(* CODESYS project AxisControl.export

Project tree, tasks and I/O mapping:
  AxisControl/
    data type MutiAxisMoveMethod
    function block AuxAxis_PowerOn [ST]
    function block MultiAxisABSMove [ST]
    function block MultiAxisTorqueLimit [ST]
*)

// AxisControl/MutiAxisMoveMethod
TYPE MutiAxisMoveMethod :
(
	None := 0				// all axis move at same vel as given
	, SpeedControl := 10		// all axis arrive destination at same time
);
END_TYPE

// AxisControl/AuxAxis_PowerOn
FUNCTION_BLOCK AuxAxis_PowerOn
VAR_INPUT
	Enable : BOOL;
END_VAR
VAR_OUTPUT
	Done : BOOL;
	Error : BOOL;
	Err_Message : Error_Message;
END_VAR
VAR
	_state : INT := 0;
	_end : BOOL := TRUE;
	_Timer: ton;
	_err_time : TIME := T#5S;
	
	// read cfg message
	ReadCfg : ArcaLibrary.SYS_GetConfigInfo;
	Num_of_Axis:WORD;
	Num_of_Groups:WORD;
	Num_of_Cams:WORD;
	MotionCfgOK: BOOL;
	ECatCfgOk: BOOL;
	VisionCfgOk: BOOL;
	
	// power settings
	PowBlk:ARRAY[1..48] OF ArcaLibrary.MC_Power;
	PowDone, PowErr: ARRAY [1..48] OF BOOL;
	power_On_States : INT := 0;
	All_Power_On_Check_Counter : INT;
	Power_Err_Check_Counter : INT;
	Power_Counter : INT;
	
	//reset blocks
	AxRes:ARRAY[1..48] OF ArcaLibrary.MC_Reset;
	AxResDone, AxResErr: ARRAY [1..48] OF BOOL;
	rest_counter : INT := 0;
	All_reset_On : BOOL;
	All_reset_On_Check_Counter : INT;
	reset_Err_Check_Counter : INT;
	reset_State : INT := 0;
	
	//group management
	GrpEn: ARRAY[1..5] OF ArcaLibrary.MC_GroupEnable;
	GrpDis: ARRAY[1..5] OF ArcaLibrary.MC_GroupDisable;
	GrpErr : ARRAY [1..5] OF BOOL;
	Grp_En_State : INT;
	Grp_counter : INT;
	Grp_En_Check_Counter : INT;
	Grp_Dis_Counter : INT;
	
	//debug
END_VAR

IF enable  THEN
	_end := FALSE;
ELSE
	_state := -10;
END_IF

IF _end = TRUE THEN
	RETURN;
END_IF

_Timer(in:= (power_On_States = 10) OR (reset_State = 10) OR (Grp_En_State = 10), pt:= _err_time);

// read how many axis has been config
ReadCfg(axisnumber => Num_of_axis, groupnumber => Num_of_Groups, cameranumber => Num_of_Cams
	, MotionCfgOk => MotionCfgOK, ecatcfgok => ECatCfgOk, visioncfgok => VisionCfgOk);

// power blocks
CASE (power_On_States) OF
	0:	
		IF (_state>0 AND _state<100) AND ECatCfgOk AND MotionCfgOK THEN
			power_On_States := 10;
		END_IF
	10:
		All_Power_On_Check_Counter := 1;
		FOR Power_Counter:=1 TO WORD_TO_INT(Num_of_axis) DO
			PowBlk[Power_Counter](Axis:=Power_Counter -1, Enable:=TRUE, EnablePositive:=TRUE, EnableNegative:=TRUE, Status=>PowDone[Power_Counter], Error=>PowErr[Power_Counter]);
			IF PowDone[Power_Counter] = TRUE THEN
				All_Power_On_Check_Counter := All_Power_On_Check_Counter + 1;
			END_IF
		END_FOR
		
		IF All_Power_On_Check_Counter >= WORD_TO_INT(Num_of_axis) THEN
			power_On_States := 20;
		ELSIF _Timer.Q THEN
			_state := -21;
		END_IF
		IF (_state<=0 OR _state>=100) THEN
			power_On_States := 30;
		END_IF
	20:
		IF (_state<=0 OR _state>=100) THEN
			power_On_States := 30;
		END_IF
	30:
		FOR Power_Counter:=1 TO WORD_TO_INT(Num_of_axis) DO
			PowBlk[Power_Counter](Axis:=Power_Counter -1, Enable:=FALSE);
		END_FOR
		power_On_States := 0;
END_CASE
// check if power block is err
IF power_On_States > 0 AND power_On_States < 30 THEN
	FOR Power_Err_Check_Counter:=1 TO WORD_TO_INT(Num_of_axis) DO
			IF PowBlk[Power_Err_Check_Counter - 1].Error = TRUE THEN
				//_state := -20;
			END_IF
	END_FOR
END_IF

// reset blocks
CASE (reset_State) OF
	0:
		All_reset_On := FALSE;
		IF _state=2 THEN
			reset_state := 10;
		END_IF
	10:
		All_reset_On_Check_Counter := 0;
		FOR rest_counter:=1 TO WORD_TO_INT(Num_of_axis) DO
			AxRes[rest_counter](Axis:=rest_counter - 1, Execute:=TRUE, Done=>AxResDone[rest_counter], Error=>AxResErr[rest_counter]);
			IF AxRes[rest_counter].Done = TRUE THEN
				All_reset_On_Check_Counter := All_reset_On_Check_Counter +1;
			END_IF
		END_FOR
		IF All_reset_On_Check_Counter = WORD_TO_INT(Num_of_axis) THEN
			All_reset_On := TRUE;
		ELSIF _Timer.Q THEN
			_state := -31;
		END_IF
		IF (_state <> 2) THEN
			reset_State := 0;
		END_IF
END_CASE
// check if reset block is err
IF reset_State <> 0 THEN
	FOR reset_Err_Check_Counter:=1 TO WORD_TO_INT(Num_of_axis) DO
			IF AxRes[reset_Err_Check_Counter - 1].Error = TRUE THEN
				_state := -30;
			END_IF
	END_FOR
END_IF

// group enable/disable
CASE Grp_En_State OF
	0:
		IF _state >= 30 AND _state <=100 THEN
			grp_counter := 1;
			Grp_En_State := 10;
		END_IF
	10:	
		IF grp_counter > WORD_TO_INT(Num_of_Groups) THEN
			Grp_En_State := 20;
		ELSE
			GrpEn[grp_counter](AxesGroup := grp_counter - 1, Execute := TRUE);
			IF GrpEn[grp_counter].Done THEN
				IF grp_counter <= WORD_TO_INT(Num_of_Groups) THEN
					grp_counter := grp_counter +1;
				END_IF
			ELSIF _Timer.Q THEN
				_state := -41;
			END_IF
		END_IF
		
		IF (_state < 30 OR _state > 100) THEN
			Grp_En_State := 30;
		END_IF
	20:
		IF (_state < 30 OR _state > 100) THEN
			Grp_En_State := 30;
		END_IF
	30:
		FOR grp_counter := 1 TO WORD_TO_INT(Num_of_Groups) DO
			GrpEn[grp_counter](AxesGroup := grp_counter - 1, Execute := FALSE);
		END_FOR
		Grp_En_State := 0;
	
END_CASE
// check if enable block is err
IF Grp_En_State = 9990 THEN
	FOR Grp_En_Check_Counter:=1 TO WORD_TO_INT(Num_of_Groups) DO
			IF GrpEn[Grp_En_Check_Counter - 1].Error = TRUE THEN
				_state := -40;
			END_IF
	END_FOR
END_IF

// disable group when all group enable block are off
FOR Grp_Dis_Counter := 1 TO WORD_TO_INT(Num_of_Groups) DO
	GrpDis[Grp_Dis_Counter](AxesGroup:= Grp_Dis_Counter - 1, Execute:= Grp_En_State = 0);
END_FOR

//	manager
CASE _state OF
	-41:
		error := TRUE;
		err_message := Error_Message.Err_Group_Enable_TimeOut;
	-40:
		error := TRUE;
		err_message := Error_Message.Err_Group_Enable_Block_Err;
		
	-31:
		error := TRUE;
		err_message := Error_Message.Err_Power_Reset_TimeOut;
	-30:
		error := TRUE;
		err_message := Error_Message.Err_Power_Reset_Block_Err;
		
	-21:
		error := TRUE;
		err_message := Error_Message.Err_PowerOn_TimeOut;
	-20:
		error := TRUE;
		err_message := Error_Message.Err_PowerOn_Block_Err;
	-10:
		IF power_On_States = 0 AND reset_State = 0 AND Grp_En_State = 0 THEN
			done := error := FALSE;
			err_message := error_message.Err_None;
			_end := TRUE;
			_state := 0;
		END_IF
	0:
		IF enable AND power_On_States = 0 AND reset_State = 0 AND Grp_En_State = 0 THEN
			_state := 10;
		END_IF
	10:
		IF power_On_States = 20 THEN
			_state := 30;
		END_IF
	30:
		IF Grp_En_State = 20 THEN
			_state := 40;
		END_IF
	40:
		done := TRUE;
END_CASE

END_FUNCTION_BLOCK

// AxisControl/MultiAxisABSMove
FUNCTION_BLOCK MultiAxisABSMove
VAR_INPUT
	FirstAuxAxisNum : BYTE;	// for safty reason, this block do not accept different axis after enabled
	LastAuxAxisNum : BYTE;
	Enable : BOOL;
	Axis_Mov_Indicator : ARRAY [0..255] OF BOOL; // tell program which axis to mov whih not mov
	Axis_Mov_Pos : ARRAY [0..255] OF REAL; // tell program which axis to what position
	Execute : BOOL;
	Vel, Acc, Dec, Jerk : REAL;	// not allow 0 or none input
	MoveMethod : MutiAxisMoveMethod;
END_VAR
VAR_OUTPUT
	done : BOOL;
	error : BOOL;
	error_str : STRING;
END_VAR
VAR
	_Faxis, _Laxis : BYTE;	// internal first axis and last axis
	_Indicator : ARRAY [0..255] OF BOOL; // internal indicator
	_enb : BOOL;
	_state : INT;
	_axisMovCmd : ARRAY [0..255] OF ArcaLibrary.MC_MoveAbsolute;
	_i : INT;
	_totalMovAxis : WORD;
	_totalMovDone : WORD;
	_err_axis : INT;
	_err_header : STRING := 'Error State: ';
	_pos : ARRAY [0..255] OF REAL;
	_speedPar : ARRAY [0..255] OF ARRAY [0..3] OF REAL;	// 255 velocity, acceleration, deceleration and jerk
	_maxDistance, _maxArriveTime : REAL;
	_readPos : ARRAY [0..255] OF ArcaLibrary.MCAT_ReadAxisMeasures;
	_currPos : ARRAY [0..255] OF REAL;
	_accRatio, _decRatio, _jerkRatio : REAL;
END_VAR


IF NOT enable THEN
	IF _enb THEN	// if local enable is turn on reset values
		FOR _i := _Faxis TO _Laxis DO	// reset all cmd block
			_axisMovCmd[_i](axis :=_i, execute := FALSE);
			_readPos[_i](axis := _i, enable := FALSE);
		END_FOR
		_enb :=
		done :=
		error := FALSE;
		delete(error_str, len := UINT_TO_INT(SIZEOF(error_str)), pos := 1);
		_state := 0;
	END_IF
	RETURN;
END_IF
IF NOT _enb THEN	// initialze
	_enb := TRUE;
	_Faxis := FirstAuxAxisNum;	// for safty reason, this block do not accept different axis after enabled
	_Laxis := LastAuxAxisNum;
	FOR _i := _Faxis TO _Laxis DO	// reset all cmd block
		_axisMovCmd[_i](axis :=_i, execute := FALSE);
	END_FOR
END_IF

CASE _state OF
	-10:
		error := TRUE;
		error_str := concat(_err_header,concat(INT_TO_STRING(_state), concat( ', Axis move block error. Error axis number is: ', INT_TO_STRING(_err_axis))));
	-2:
		error := TRUE;
		error_str := concat(_err_header,concat(INT_TO_STRING(_state), ', speed parameter input is 0'));
	-1:
		error := TRUE;
		error_str := concat(_err_header,concat(INT_TO_STRING(_state), ', there are no such MoveMethod as given'));
	0:
		IF execute THEN
			IF vel = 0 OR acc = 0 OR dec = 0 OR jerk = 0 THEN
				_state := -2;
				RETURN;
			END_IF
			_pos := Axis_Mov_Pos;	// transfer to local value for safe
			_Indicator := Axis_Mov_Indicator;
			CASE MoveMethod OF
				0:	
					FOR _i := _Faxis TO _Laxis DO
						_speedPar[_i][0] := vel;
						_speedPar[_i][1] := acc;
						_speedPar[_i][2] := dec;
						_speedPar[_i][3] := jerk;
					END_FOR
				10:	// calculate all axis insure them arrive destination
					_accRatio := acc/vel;	// accRaito
					_decRatio := dec/vel;	// decRaito
					_jerkRatio := jerk/acc;	// JerkaRito
					FOR _i := _Faxis TO _Laxis DO	// find which axis have most far destination
						IF _Indicator[_i] THEN
							_readPos[_i](axis := _i, enable := TRUE, pos => _currPos[_i]);
							IF _maxDistance < ABS(_currPos[_i] - _pos[_i]) THEN
								_maxDistance := ABS(_currPos[_i] - _pos[_i]);
							END_IF
							_readPos[_i](axis := _i, enable := FALSE);
						END_IF
					END_FOR
					_maxArriveTime := _maxDistance/vel;
					FOR _i := _Faxis TO _Laxis DO	// calculate individual speed parameter for each axis
						IF _Indicator[_i] THEN
							_speedPar[_i][0] := ABS(_currPos[_i] - _pos[_i])/_maxArriveTime;
							_speedPar[_i][1] := _speedPar[_i][0] * _accRatio;
							_speedPar[_i][2] := _speedPar[_i][0] * _decRatio;
							_speedPar[_i][3] := _speedPar[_i][1] * _jerkRatio;
						END_IF
					END_FOR
			ELSE
				error := TRUE;
				_state := -1;
				RETURN;
			END_CASE
			_state := 10;
		END_IF
	10:
		_totalMovAxis := _totalMovDone := 0;
		_i := _Faxis;
		
		WHILE _i <= _Laxis AND NOT error DO
			IF _Indicator[_i] THEN	// if indicator show _i motor need to be command
				_axisMovCmd[_i](axis := _i, execute := TRUE, Position := _pos[_i]
					, velocity := _speedPar[_i][0], acceleration := _speedPar[_i][1], Deceleration := _speedPar[_i][2], Jerk := _speedPar[_i][3]
					, Direction := mcShortestway, Buffermode := mcAborting);
				_totalMovAxis := _totalMovAxis + 1;	// count how many axis are indicate to move
				IF _axisMovCmd[_i].Done THEN
					_totalMovDone := _totalMovDone + 1;
				END_IF
				IF _axisMovCmd[_i].Error THEN
					error := TRUE;
					_err_axis := _i;
				END_IF
			END_IF
			_i := _i + 1;
		END_WHILE
		IF error THEN
			_state := -10;
		ELSIF NOT error AND _totalMovAxis = _totalMovDone THEN	// all axis move done and no error
			FOR _i := _Faxis TO _Laxis DO	// reset all cmd block
				_axisMovCmd[_i](axis :=_i, execute := FALSE);
			END_FOR
			done := TRUE;
			_state := 20;
		END_IF
	20:
		IF NOT execute THEN
			done := FALSE;
			_state := 0;
		END_IF
END_CASE

// debug

_axisMovCmd[00].Done;
_axisMovCmd[01].Done;
_axisMovCmd[02].Done;
_axisMovCmd[03].Done;
_axisMovCmd[04].Done;
_axisMovCmd[05].Done;
_axisMovCmd[06].Done;
_axisMovCmd[07].Done;
_axisMovCmd[08].Done;
_axisMovCmd[09].Done;
_axisMovCmd[10].Done;
_axisMovCmd[11].Done;
_axisMovCmd[12].Done;
_axisMovCmd[13].Done;
_axisMovCmd[14].Done;
_axisMovCmd[15].Done;
_axisMovCmd[16].Done;
_axisMovCmd[17].Done;

END_FUNCTION_BLOCK

// AxisControl/MultiAxisTorqueLimit
FUNCTION_BLOCK MultiAxisTorqueLimit
VAR_INPUT
	FirstAuxAxisNum : BYTE;	// for safty reason, this block do not accept different axis after enabled
	LastAuxAxisNum : BYTE;
	Enable : BOOL;
	Axis_Torque_Limit_Indicator : ARRAY [0..255] OF BOOL; // tell program which axis to limit Torque
	Axis_Torque_Limit_Value : ARRAY [0..255] OF REAL; // tell program which axis's torque limition
	Execute : BOOL;
END_VAR
VAR_OUTPUT
	done : BOOL;
	error : BOOL;
	error_str : STRING;
END_VAR
VAR
	_Faxis, _Laxis : BYTE;	// internal first axis and last axis
	_indicator : ARRAY [0..255] OF BOOL; // internal torque indicator
	_enb : BOOL;
	_state : INT;
	_axisLimitionCmd : ARRAY [0..255] OF ArcaLibrary.MCAT_AxisSetLimits;
	_i : INT;
	_totalNeedSetAxis : WORD;
	_totalSetDone : WORD;
	_err_axis : INT;
	_err_header : STRING := 'Error State: ';

	_toque_limit : ARRAY [0..255] OF REAL;
	
END_VAR


IF NOT enable THEN
	IF _enb THEN	// if local enable is turn on reset values
		FOR _i := _Faxis TO _Laxis DO	// reset all cmd block
			_axisLimitionCmd[_i](axis :=_i, execute := FALSE);
		END_FOR
		_enb :=
		done :=
		error := FALSE;
		delete(error_str, len := UINT_TO_INT(SIZEOF(error_str)), pos := 1);
		_state := 0;
	END_IF
	RETURN;
END_IF
IF NOT _enb THEN	// initialze
	_enb := TRUE;
	_Faxis := FirstAuxAxisNum;	// for safty reason, this block do not accept different axis after enabled
	_Laxis := LastAuxAxisNum;
	FOR _i := _Faxis TO _Laxis DO	// reset all cmd block
		_axisLimitionCmd[_i](axis :=_i, execute := FALSE);
	END_FOR
END_IF

CASE _state OF
	-10:
		error := TRUE;
		error_str := concat(_err_header,concat(INT_TO_STRING(_state), concat( ', Axis move block error. Error axis number is: ', INT_TO_STRING(_err_axis))));
	-1:
		error := TRUE;
		error_str := concat(_err_header,concat(INT_TO_STRING(_state), ', there are no such MoveMethod as given'));
	0:
		IF execute THEN
			_toque_limit := Axis_Torque_Limit_Value;	// transfer to local value for safe
			_indicator := Axis_Torque_Limit_Indicator;
			_state := 10;
		END_IF
	10:
		_totalSetDone := _totalNeedSetAxis := 0;
		_i := _Faxis;
		
		WHILE _i <= _Laxis AND NOT error DO
			IF _indicator[_i] THEN	// if indicator show _i motor need to be command
				_axisLimitionCmd[_i](axis := _i, execute := TRUE, TorqueLimit := _toque_limit[_i]);
				_totalNeedSetAxis := _totalNeedSetAxis + 1;	// count how many axis are indicate to move
				IF _axisLimitionCmd[_i].Done THEN
					_totalSetDone := _totalSetDone + 1;
				END_IF
				IF _axisLimitionCmd[_i].Error THEN
					error := TRUE;
					_err_axis := _i;
				END_IF
			END_IF
			_i := _i + 1;
		END_WHILE
		IF error THEN
			_state := -10;
		ELSIF NOT error AND _totalNeedSetAxis = _totalSetDone THEN	// all axis move done and no error
			FOR _i := _Faxis TO _Laxis DO	// reset all cmd block
				_axisLimitionCmd[_i](axis :=_i, execute := FALSE);
			END_FOR
			done := TRUE;
			_state := 20;
		END_IF
	20:
		IF NOT execute THEN
			done := FALSE;
			_state := 0;
		END_IF
END_CASE

END_FUNCTION_BLOCK
